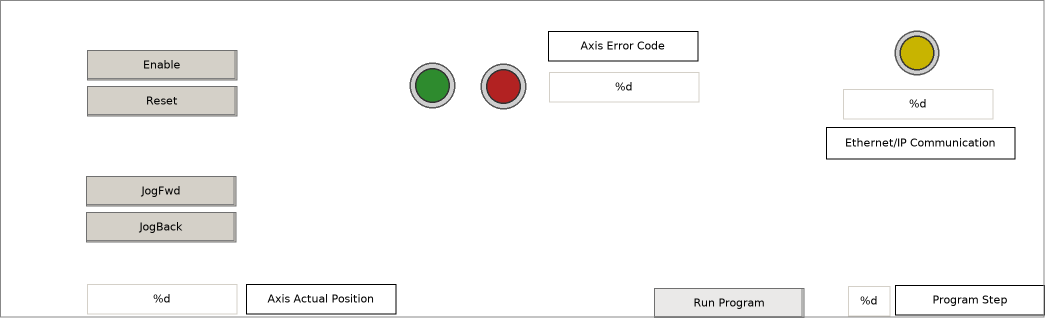
VISUALIZATION Visualization  // 1045x318
    Button (86,176 150x30), "JogFwd"
        OnMouseDown: toggle MAIN.TwinCAT_jogFwd
        OnMouseUp: toggle MAIN.TwinCAT_jogFwd
    Button (86,212 150x30), "JogBack"
        OnMouseDown: toggle MAIN.TwinCAT_jogBack
        OnMouseUp: toggle MAIN.TwinCAT_jogBack
    Lamp1 (406,57 53x57), variable: MAIN.bEnable, style: Lamp-Lamp1-Green
    Lamp1 (477,59 53x55), variable: MAIN.bError, style: Lamp-Lamp1-Red
    Button (87,50 150x30), "Enable"
        OnMouseDown: toggle MAIN.TwinCAT_bEnable
    Button (87,86 150x30), "Reset"
        OnMouseDown: toggle MAIN.TwinCAT_bReset
        OnMouseUp: toggle MAIN.TwinCAT_bReset
    Lamp1 (891,27 52x52), variable: MAIN.LinkError, style: Lamp-Lamp1-Yellow
    Textfield (843,89 150x30), "%d", text variable: MAIN.AB_Connected
    Textfield (549,72 150x30), "%d", text variable: MAIN.DriveErrorCode
    Textfield (87,284 150x30), "%d", text variable: MAIN.Axis1.NcToPlc.ActPos
    Button (654,288 150x30), "Run Program", colour toggle: MAIN.TwinCAT_StartProgram
        OnMouseDown: toggle MAIN.TwinCAT_StartProgram
    Textfield (848,286 42x30), "%d", text variable: MAIN.ProgramStep
    Rectangle (548,31 150x30), "Axis Error Code"
    Rectangle (826,127 189x32), "Ethernet/IP Communication"
    Rectangle (246,284 150x30), "Axis Actual Position"
    Rectangle (895,285 150x30), "Program Step"
END_VISUALIZATION

(* stored: Version 1.1.0.1, ProductVersion 3.1.4024.12
   Visu Visualization: Id {e7124508-ac53-491e-9a0f-c456c71fc0d3} *)
